// TwinCAT 3 PLC project PLC_Student
// ProgramVersion: 3.1.4024.0
// libraries:
//   Tc2_Standard, * (Beckhoff Automation GmbH)
//   Tc2_System, * (Beckhoff Automation GmbH)
//   Tc3_Module, * (Beckhoff Automation GmbH)
// project tree:
//   / GlobalTextList.TcGTLO, PlcTask.TcTTO, Visualization Manager.TcVMO (not stored)
//   GVLs/ GVL.TcGVL
//   POUs/ Control_SFC.TcPOU, MAIN.TcPOU
//   VISUs/ Visualization.TcVIS
// (motion and I/O tree: see PLC project plc_sim)
// real-time tasks:
//   TASK PlcTask: cycle T#10ms, priority 20, ADS port 350
//   TASK PlcTask1: cycle T#10ms, priority 21, ADS port 351
// variable links:
//   PLC_Sim/PLC_Sim Instance <-> PLC_Student/PLC_Student Instance
//     PlcTask Inputs/GVL.ixDir <-> PlcTask Outputs/GVL.qxDir
//     PlcTask Inputs/GVL.ixStrobe <-> PlcTask Outputs/GVL.qxStrobe
//     PlcTask Outputs/GVL.qiAtStation1 <-> PlcTask Inputs/GVL.iiAtStation1
//     PlcTask Outputs/GVL.qiAtStation2 <-> PlcTask Inputs/GVL.iiAtStation2

CONFIGURATION PLC_Student
    RESOURCE PLC ON TwinCAT3
        TASK PlcTask(INTERVAL := T#10ms, PRIORITY := 21);
        PROGRAM MAIN WITH PlcTask : MAIN;
    END_RESOURCE
END_CONFIGURATION

// ---- GVLs/GVL.TcGVL
{attribute 'qualified_only'}
VAR_GLOBAL
//Output from process to PLC
	qxStrobe		AT %Q*:	BOOL;
	qxDir			AT %Q*:	INT;
	
//Input to process from PLC
	iiAtStation1		AT %I*:	BOOL;
	iiAtStation2		AT %I*:	BOOL;
END_VAR

// ---- POUs/MAIN.TcPOU
PROGRAM MAIN
VAR
END_VAR

Control_SFC();

END_PROGRAM

// ---- POUs/Control_SFC.TcPOU
PROGRAM Control_SFC
VAR
	iSetManual: BOOL;
	iSetAuto: BOOL;
	iAutoStart: BOOL;
	iManualLeft: BOOL;
	iManualRight: BOOL;
	iAutoStop: BOOL;
	iStop: BOOL;
	
	xMode: STRING;
	xAutomatic: BOOL;
	xManual: BOOL;
	xAutoStart: BOOL;
	xAutoStop: BOOL;
	xManualLeft: BOOL;
	xManualRight: BOOL;
END_VAR

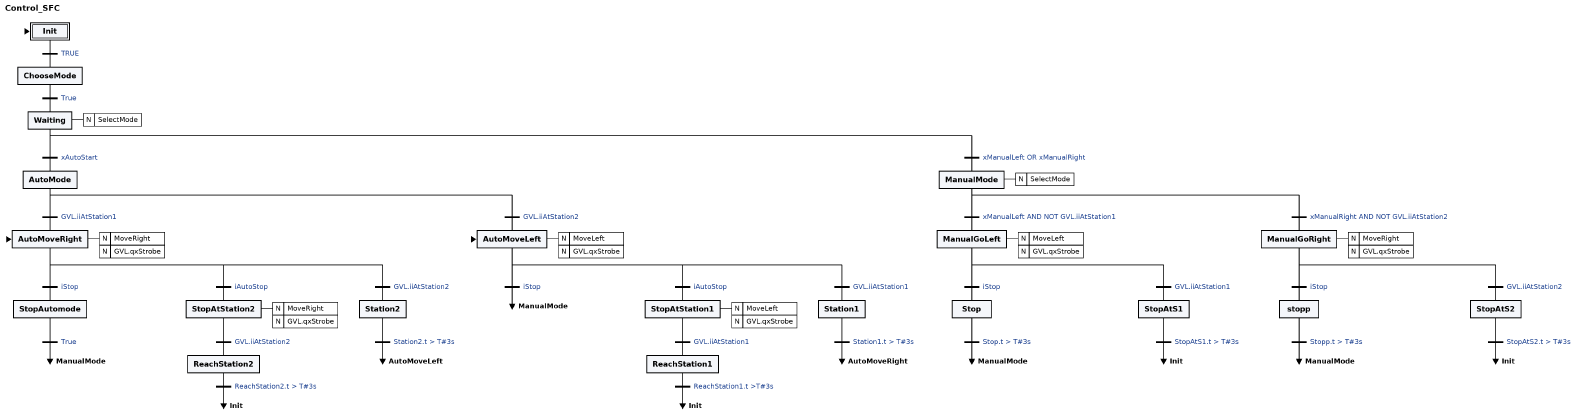
INITIAL_STEP Init:
END_STEP
TRANSITION FROM Init TO ChooseMode
    := TRUE;
END_TRANSITION
STEP ChooseMode:
END_STEP
TRANSITION FROM ChooseMode TO Waiting
    := True;
END_TRANSITION
STEP Waiting:
    SelectMode(N);
END_STEP
TRANSITION FROM Waiting TO AutoMode
    := xAutoStart;
END_TRANSITION
STEP AutoMode:
END_STEP
TRANSITION FROM AutoMode TO AutoMoveRight
    := GVL.iiAtStation1;
END_TRANSITION
STEP AutoMoveRight:
    MoveRight(N);
    GVL.qxStrobe(N);
END_STEP
TRANSITION FROM AutoMoveRight TO StopAutomode
    := iStop;
END_TRANSITION
STEP StopAutomode:
END_STEP
TRANSITION FROM StopAutomode TO ManualMode
    := True;
END_TRANSITION
TRANSITION FROM AutoMoveRight TO StopAtStation2
    := iAutoStop;
END_TRANSITION
TRANSITION FROM AutoMoveRight TO Station2
    := GVL.iiAtStation2;
END_TRANSITION
STEP Station2:
END_STEP
TRANSITION FROM Station2 TO AutoMoveLeft
    := Station2.t > T#3s;
END_TRANSITION
STEP StopAtStation2:
    MoveRight(N);
    GVL.qxStrobe(N);
END_STEP
TRANSITION FROM StopAtStation2 TO ReachStation2
    := GVL.iiAtStation2;
END_TRANSITION
STEP ReachStation2:
END_STEP
TRANSITION FROM ReachStation2 TO Init
    := ReachStation2.t > T#3s;
END_TRANSITION
TRANSITION FROM AutoMode TO AutoMoveLeft
    := GVL.iiAtStation2;
END_TRANSITION
STEP AutoMoveLeft:
    MoveLeft(N);
    GVL.qxStrobe(N);
END_STEP
TRANSITION FROM AutoMoveLeft TO ManualMode
    := iStop;
END_TRANSITION
TRANSITION FROM AutoMoveLeft TO StopAtStation1
    := iAutoStop;
END_TRANSITION
TRANSITION FROM AutoMoveLeft TO Station1
    := GVL.iiAtStation1;
END_TRANSITION
STEP Station1:
END_STEP
TRANSITION FROM Station1 TO AutoMoveRight
    := Station1.t > T#3s;
END_TRANSITION
STEP StopAtStation1:
    MoveLeft(N);
    GVL.qxStrobe(N);
END_STEP
TRANSITION FROM StopAtStation1 TO ReachStation1
    := GVL.iiAtStation1;
END_TRANSITION
STEP ReachStation1:
END_STEP
TRANSITION FROM ReachStation1 TO Init
    := ReachStation1.t >T#3s;
END_TRANSITION
TRANSITION FROM Waiting TO _ManualMode
    := xManualLeft OR xManualRight;
END_TRANSITION
STEP _ManualMode:  // name as stored:  ManualMode
    SelectMode(N);
END_STEP
TRANSITION FROM _ManualMode TO ManualGoLeft
    := xManualLeft AND NOT GVL.iiAtStation1;
END_TRANSITION
STEP ManualGoLeft:
    MoveLeft(N);
    GVL.qxStrobe(N);
END_STEP
TRANSITION FROM ManualGoLeft TO Stop
    := iStop;
END_TRANSITION
STEP Stop:
END_STEP
TRANSITION FROM Stop TO ManualMode
    := Stop.t > T#3s;
END_TRANSITION
TRANSITION FROM ManualGoLeft TO StopAtS1
    := GVL.iiAtStation1;
END_TRANSITION
STEP StopAtS1:
END_STEP
TRANSITION FROM StopAtS1 TO Init
    := StopAtS1.t > T#3s;
END_TRANSITION
TRANSITION FROM _ManualMode TO ManualGoRight
    := xManualRight AND NOT GVL.iiAtStation2;
END_TRANSITION
STEP ManualGoRight:
    MoveRight(N);
    GVL.qxStrobe(N);
END_STEP
TRANSITION FROM ManualGoRight TO stopp
    := iStop;
END_TRANSITION
STEP stopp:
END_STEP
TRANSITION FROM stopp TO ManualMode
    := Stopp.t > T#3s;
END_TRANSITION
TRANSITION FROM ManualGoRight TO StopAtS2
    := GVL.iiAtStation2;
END_TRANSITION
STEP StopAtS2:
END_STEP
TRANSITION FROM StopAtS2 TO Init
    := StopAtS2.t > T#3s;
END_TRANSITION

ACTION MoveLeft:
GVL.qxDir := -1;
END_ACTION

ACTION MoveRight:
GVL.qxDir := 1;
END_ACTION

ACTION SelectMode:
xAutoStart := FALSE;
xAutoStop := FALSE;
xManualLeft := FALSE;
xManualRight := FALSE;

IF iSetManual THEN
	xAutomatic := FALSE;
	xManual := TRUE;
	xMode := 'Manual';
ELSIF iSetAuto THEN 
	xAutomatic := TRUE;
	xManual := FALSE;
	xMode := 'Automatic';
END_IF

IF xAutomatic THEN
	IF iAutoStart THEN
		xAutoStart := TRUE;
		xAutoStop := FALSE;
	ELSIF iAutoStop THEN
		xAutoStart := FALSE;
		xAutoStop := TRUE;
	END_IF
END_IF

IF xManual THEN
	IF iManualLeft THEN
		xManualLeft := TRUE;
		xManualRight := FALSE;
	ELSIF iManualRight THEN
		xManualLeft := FALSE;
		xManualRight := TRUE;
	END_IF
END_IF
END_ACTION

END_PROGRAM

// ---- GlobalTextList.TcGTLO
TEXTLIST GlobalTextList
  214 = '%s'
  489 = 'Auto Start'
  734 = 'Auto Stop'
  899 = 'Automatic Mode'
  938 = 'Automatic Start'
  358 = 'Emergency Stop'
  66 = 'Go automatic'
  433 = 'Go Left'
  265 = 'Go left'
  347 = 'Go Right'
  549 = 'khj'
  24 = 'Manual Backward'
  241 = 'Manual Forward'
  531 = 'Manual Left'
  670 = 'Manual Mode'
  649 = 'Manual Right'
  366 = 'sdf'
  541 = 'Set Auto'
  286 = 'Set Automatic'
  437 = 'Set Manual'
  243 = 'Set Manuals'
  288 = 'Start'
  892 = 'Start Auto'
  572 = 'Stop'
  152 = 'Stop Auto'
  293 = 'Towards Left'
  886 = 'Towards Right'
  882 = 'Towards Station1'
  875 = 'Towards Station2'
END_TEXTLIST

// ---- VISUs/Visualization.TcVIS
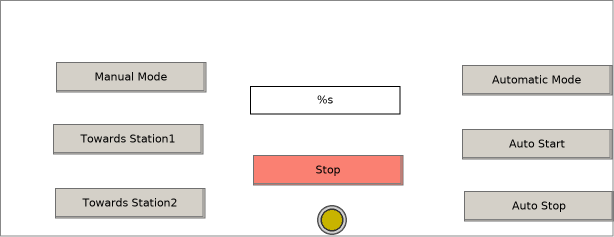
VISUALIZATION Visualization  // 614x237
    Button (56,62 150x30), "Manual Mode"
        tap Control_SFC.iSetManual
    Button (53,124 150x30), "Towards Station1"
        tap Control_SFC.iManualLeft
    Button (55,188 150x30), "Towards Station2"
        tap Control_SFC.iManualRight
    Button (462,65 150x30), "Automatic Mode"
        tap Control_SFC.iSetAuto
    Button (462,129 150x30), "Auto Start"
        tap Control_SFC.iAutoStart
    Button (464,191 150x30), "Auto Stop"
        tap Control_SFC.iAutoStop
    Button (253,155 150x30), "Stop"
        tap Control_SFC.iStop
    Rectangle (250,86 150x28), "%s", text variable: Control_SFC.xMode
    Lamp1 (311,203 42x34), style: Lamp-Lamp1-Yellow
END_VISUALIZATION
